SUBAPPLICATION mapping_Uebung_026 (* Spiegelabfolge (6) *)
  (* Standard: 61499-2; Description: Copyright (c) 2023 Meisterschulen am Ostbahnhof This program and the accompanying materials are made available under the terms of the Eclipse Public License 2.0 which is available at https://www.eclipse.org/legal/epl-2.0/ SPDX-License-Identifier: EPL-2.0 *)
  (* Version 1.0, 2023-10-23, Franz Höpfinger, Meisterschulen am Ostbahnhof *)
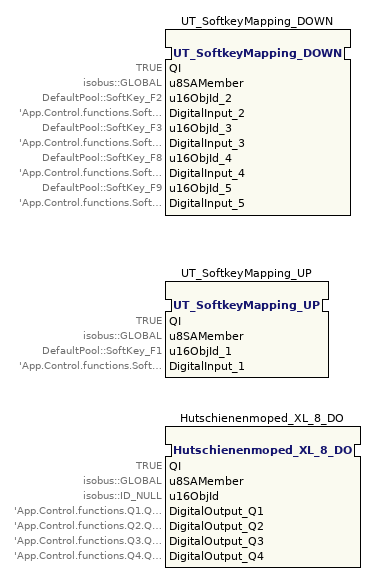
  FBS
    Hutschienenmoped_XL_8_DO : Hutschienenmoped_XL_8_DO(QI := TRUE, u8SAMember := isobus::GLOBAL, u16ObjId := isobus::ID_NULL, DigitalOutput_Q1 := 'App.Control.functions.Q1.QX', DigitalOutput_Q2 := 'App.Control.functions.Q2.QX', DigitalOutput_Q3 := 'App.Control.functions.Q3.QX', DigitalOutput_Q4 := 'App.Control.functions.Q4.QX');
    UT_SoftkeyMapping_UP : UT_SoftkeyMapping_UP(QI := TRUE, u8SAMember := isobus::GLOBAL, u16ObjId_1 := DefaultPool::SoftKey_F1, DigitalInput_1 := 'App.Control.functions.SoftKey_F1_UP');
    UT_SoftkeyMapping_DOWN : UT_SoftkeyMapping_DOWN(QI := TRUE, u8SAMember := isobus::GLOBAL, u16ObjId_2 := DefaultPool::SoftKey_F2, DigitalInput_2 := 'App.Control.functions.SoftKey_F2_DOWN', u16ObjId_3 := DefaultPool::SoftKey_F3, DigitalInput_3 := 'App.Control.functions.SoftKey_F3_DOWN', u16ObjId_4 := DefaultPool::SoftKey_F8, DigitalInput_4 := 'App.Control.functions.SoftKey_F8_DOWN', u16ObjId_5 := DefaultPool::SoftKey_F9, DigitalInput_5 := 'App.Control.functions.SoftKey_F9_DOWN');
  END_FBS
END_SUBAPPLICATION
